// TIA Portal V17 export
// export: Created 2024-09-02T12:50:34.177996Z, ExportSetting WithDefaults, DisplayName Totally Integrated Automation Portal, DisplayVersion V17, DisplayName TIA Portal Openness, DisplayVersion V17, DisplayName TIA Portal Version Control Interface, DisplayVersion V17, DisplayName STEP 7 Professional, DisplayVersion V17, DisplayName STEP 7 Safety, DisplayVersion V17, DisplayName WinCC Professional, DisplayVersion V17
TYPE "typ_MobyDMCTaf"
// stored: IsFailsafeCompliant false
   STRUCT
      DMC { ExternalWritable := 'False'; S7_SetPoint := 'True'} : Array[1..8] of "typ_MobyDMC";
   END_STRUCT;
END_TYPE
